(* CODESYS project e!C_Integration_Test_1.ECP

Project tree, tasks and I/O mapping:
  PFC200_CS_2ETH_RS_CAN_DPS : 750-8206 PFC200 2ETH RS CAN DPS, WAGO, order no. 0750-8206, version 5.11.1.16
    application PFC8206
      libraries: Util, * (System); VisuDialogs, * (System)
      task PLC_Task (cyclic, interval t#10ms, priority 14) calls PLC_PRG
      task VISU_TASK (cyclic, interval 100 ms, priority 15) calls VisuElems.Visu_Prg
      task AlarmManagerTask (cyclic, interval 50 ms, priority 15) calls AlarmManager.Alarm_Prg
      program PLC_PRG [ST]: BlinkTest1, Modbus, NetVar
      visualisation Visu1
      Alarm_Configuration
        alarm class Error (priority 10, acknowledge REP_ACK)
        alarm class Warning (priority 30, acknowledge REP)
        alarm class Info (priority 100, acknowledge REP)
        AlarmStorage
        text list AlarmGroup1
        alarm group AlarmGroup1
            0 [Error]: Comparison Equal, ExpressionToCompare TRUE, Expression DO1 - "MinAlarm1"
      Scaling/
        function block fbScale_AI_455 [ST]
        function block fbScale_AI_457 [ST]
        function block fbScale_AI_457_Positiv [ST]
        function block fbScale_AI_460 [ST]
        function block fbScale_AI_461 [ST]
        function block fbScale_AI_466 [ST]
        function block fbScale_AI_473 [ST]
        function block fbScale_AO_552 [ST]
        function block fbScale_AO_555 [ST]
        function block fbScale_AO_556 [ST]
        function block fbScale_AO_559 [ST]
      program ScaleTest [CFC]: AnalogInput, AnalogOutput
      MODBUS/
        data type typFC352_tcp
        data type typPFC200_CS_2ETH_CAN_tcpPFC8203PLC_PRG
        data type typPFC200_CS_2ETH_CAN_tcpPFC8203
        data type typPFC200_CS_2ETH_CAN_tcp
      global variables MODBUS
      global variables NVL1_From_8206
      declarations NVL1_From_8203
    DeviceAdapter
    CANbus
      WAGO_CANopen_Manager : WAGO CANopen Manager, WAGO, version 3.5.4.10
          settings: ConfigVersion = 50659584
        _750_347m_V14 : 750-347m_V14, WAGO, order no. 750-347, version Revision=16#00000001, FileVersion=1.14
            settings: General Options.Reset Node = false; NODEIDSAVED = 5; SDO Timeout = 1000000; SubIndex for reset node = 0; Emergency-General Parameters.Emergency COBID = 16#00000085; Settings.COBID = 16#00000205; Settings.Transmission Type = 16#FF; Settings.available PDO-Parameter.Inhibit Time available = FALSE; Settings.available PDO-Parameter.Event Timer available = FALSE; Settings.Inhibit Time = 0; Settings.Event Timer = 0; Generic COBID = '$NODEID+16#0200'; Process by CANopenManager = TRUE; Settings.COBID = 16#00000185; Settings.Transmission Type = 16#FF; Settings.available PDO-Parameter.Inhibit Time available = TRUE; Settings.available PDO-Parameter.Event Timer available = TRUE; Settings.Inhibit Time = 0; Settings.Event Timer = 0; Generic COBID = '$NODEID+16#0180'; Process by CANopenManager = TRUE; N/A.Index = 16#6200; N/A.Subindex = 16#01; N/A.ObjectLength = 8; N/A.Index = 16#6401; N/A.Subindex = 16#01; N/A.ObjectLength = 16; N/A.Index = 16#6401; N/A.Subindex = 16#02; N/A.ObjectLength = 16; N/A.Index = 16#6401; N/A.Subindex = 16#03; N/A.ObjectLength = 16; N/A.Index = 16#6401; N/A.Subindex = 16#04; N/A.ObjectLength = 16; SDO List.Set Guardtime.Index = 16#100C; SDO List.Set Guardtime.Subindex = 16#00; SDO List.Set Guardtime.Value = 16#00000000; SDO List.Set Guardtime.Size = 16;
              SDO List.Set Guardtime.AbortIfError = FALSE; SDO List.Set Guardtime.JumpToLine = FALSE; SDO List.Set Guardtime.Line = 0; SDO List.Set Lifetime.Index = 16#100D; SDO List.Set Lifetime.Subindex = 16#00; SDO List.Set Lifetime.Value = 16#00000000; SDO List.Set Lifetime.Size = 8; SDO List.Set Lifetime.AbortIfError = FALSE; SDO List.Set Lifetime.JumpToLine = FALSE; SDO List.Set Lifetime.Line = 0; SDO List.Disable Emcy CobID.Index = 16#1014; SDO List.Disable Emcy CobID.Subindex = 16#00; SDO List.Disable Emcy CobID.Value = 16#80000085; SDO List.Disable Emcy CobID.Size = 32; SDO List.Disable Emcy CobID.AbortIfError = FALSE; SDO List.Disable Emcy CobID.JumpToLine = FALSE; SDO List.Disable Emcy CobID.Line = 0; SDO List.Set Emcy CobID.Index = 16#1014; SDO List.Set Emcy CobID.Subindex = 16#00; SDO List.Set Emcy CobID.Value = 16#00000085; SDO List.Set Emcy CobID.Size = 32; SDO List.Set Emcy CobID.AbortIfError = FALSE; SDO List.Set Emcy CobID.JumpToLine = FALSE; SDO List.Set Emcy CobID.Line = 0; SDO List.Set Heartbeat Consumer.Index = 16#1016; SDO List.Set Heartbeat Consumer.Subindex = 16#01; SDO List.Set Heartbeat Consumer.Value = 0; SDO List.Set Heartbeat Consumer.Size = 32; SDO List.Set Heartbeat Consumer.AbortIfError = FALSE; SDO List.Set Heartbeat Consumer.JumpToLine = FALSE; SDO List.Set Heartbeat Consumer.Line = 0; SDO List.Set Heartbeat Consumer.Index = 16#1016; SDO List.Set Heartbeat Consumer.Subindex = 16#02; SDO List.Set Heartbeat Consumer.Value = 0; SDO List.Set Heartbeat Consumer.Size = 32; SDO List.Set Heartbeat Consumer.AbortIfError = FALSE; SDO List.Set Heartbeat Consumer.JumpToLine = FALSE; SDO List.Set Heartbeat Consumer.Line = 0; SDO List.Set Heartbeat Consumer.Index = 16#1016; SDO List.Set Heartbeat Consumer.Subindex = 16#03;
              SDO List.Set Heartbeat Consumer.Value = 0; SDO List.Set Heartbeat Consumer.Size = 32; SDO List.Set Heartbeat Consumer.AbortIfError = FALSE; SDO List.Set Heartbeat Consumer.JumpToLine = FALSE; SDO List.Set Heartbeat Consumer.Line = 0; SDO List.Set Heartbeat Consumer.Index = 16#1016; SDO List.Set Heartbeat Consumer.Subindex = 16#04; SDO List.Set Heartbeat Consumer.Value = 0; SDO List.Set Heartbeat Consumer.Size = 32; SDO List.Set Heartbeat Consumer.AbortIfError = FALSE; SDO List.Set Heartbeat Consumer.JumpToLine = FALSE; SDO List.Set Heartbeat Consumer.Line = 0; SDO List.Set Heartbeat Consumer.Index = 16#1016; SDO List.Set Heartbeat Consumer.Subindex = 16#05; SDO List.Set Heartbeat Consumer.Value = 0; SDO List.Set Heartbeat Consumer.Size = 32; SDO List.Set Heartbeat Consumer.AbortIfError = FALSE; SDO List.Set Heartbeat Consumer.JumpToLine = FALSE; SDO List.Set Heartbeat Consumer.Line = 0; SDO List.Set Heartbeat Producer.Index = 16#1017; SDO List.Set Heartbeat Producer.Subindex = 16#00; SDO List.Set Heartbeat Producer.Value = 16#00000000; SDO List.Set Heartbeat Producer.Size = 16; SDO List.Set Heartbeat Producer.AbortIfError = FALSE; SDO List.Set Heartbeat Producer.JumpToLine = FALSE; SDO List.Set Heartbeat Producer.Line = 0; SDO List.Disable PDO.Index = 16#1400; SDO List.Disable PDO.Subindex = 16#01; SDO List.Disable PDO.Value = 16#80000205; SDO List.Disable PDO.Size = 32; SDO List.Disable PDO.AbortIfError = FALSE; SDO List.Disable PDO.JumpToLine = FALSE; SDO List.Disable PDO.Line = 0; SDO List.Set transmission type.Index = 16#1400; SDO List.Set transmission type.Subindex = 16#02; SDO List.Set transmission type.Value = 16#FF; SDO List.Set transmission type.Size = 8; SDO List.Set transmission type.AbortIfError = FALSE; SDO List.Set transmission type.JumpToLine = FALSE; SDO List.Set transmission type.Line = 0;
              SDO List.Clear pdo mapping.Index = 16#1600; SDO List.Clear pdo mapping.Subindex = 16#00; SDO List.Clear pdo mapping.Value = 16#0; SDO List.Clear pdo mapping.Size = 8; SDO List.Clear pdo mapping.AbortIfError = FALSE; SDO List.Clear pdo mapping.JumpToLine = FALSE; SDO List.Clear pdo mapping.Line = 0; SDO List.Set Mapping.Index = 16#1600; SDO List.Set Mapping.Subindex = 16#01; SDO List.Set Mapping.Value = 16#62000108; SDO List.Set Mapping.Size = 32; SDO List.Set Mapping.AbortIfError = FALSE; SDO List.Set Mapping.JumpToLine = FALSE; SDO List.Set Mapping.Line = 0; SDO List.Set number of mappings.Index = 16#1600; SDO List.Set number of mappings.Subindex = 16#00; SDO List.Set number of mappings.Value = 16#01; SDO List.Set number of mappings.Size = 8; SDO List.Set number of mappings.AbortIfError = FALSE; SDO List.Set number of mappings.JumpToLine = FALSE; SDO List.Set number of mappings.Line = 0; SDO List.Set and enable COB-ID.Index = 16#1400; SDO List.Set and enable COB-ID.Subindex = 16#01; SDO List.Set and enable COB-ID.Value = 16#00000205; SDO List.Set and enable COB-ID.Size = 32; SDO List.Set and enable COB-ID.AbortIfError = FALSE; SDO List.Set and enable COB-ID.JumpToLine = FALSE; SDO List.Set and enable COB-ID.Line = 0; SDO List.Disable PDO.Index = 16#1800; SDO List.Disable PDO.Subindex = 16#01; SDO List.Disable PDO.Value = 16#80000185; SDO List.Disable PDO.Size = 32; SDO List.Disable PDO.AbortIfError = FALSE; SDO List.Disable PDO.JumpToLine = FALSE; SDO List.Disable PDO.Line = 0; SDO List.Set transmission type.Index = 16#1800; SDO List.Set transmission type.Subindex = 16#02; SDO List.Set transmission type.Value = 16#FF; SDO List.Set transmission type.Size = 8; SDO List.Set transmission type.AbortIfError = FALSE;
              SDO List.Set transmission type.JumpToLine = FALSE; SDO List.Set transmission type.Line = 0; SDO List.Set inhibit time.Index = 16#1800; SDO List.Set inhibit time.Subindex = 16#03; SDO List.Set inhibit time.Value = 16#0000; SDO List.Set inhibit time.Size = 16; SDO List.Set inhibit time.AbortIfError = FALSE; SDO List.Set inhibit time.JumpToLine = FALSE; SDO List.Set inhibit time.Line = 0; SDO List.Set event time.Index = 16#1800; SDO List.Set event time.Subindex = 16#05; SDO List.Set event time.Value = 16#0000; SDO List.Set event time.Size = 16; SDO List.Set event time.AbortIfError = FALSE; SDO List.Set event time.JumpToLine = FALSE; SDO List.Set event time.Line = 0; SDO List.Clear pdo mapping.Index = 16#1A00; SDO List.Clear pdo mapping.Subindex = 16#00; SDO List.Clear pdo mapping.Value = 16#0; SDO List.Clear pdo mapping.Size = 8; SDO List.Clear pdo mapping.AbortIfError = FALSE; SDO List.Clear pdo mapping.JumpToLine = FALSE; SDO List.Clear pdo mapping.Line = 0; SDO List.Set Mapping.Index = 16#1A00; SDO List.Set Mapping.Subindex = 16#01; SDO List.Set Mapping.Value = 16#64010110; SDO List.Set Mapping.Size = 32; SDO List.Set Mapping.AbortIfError = FALSE; SDO List.Set Mapping.JumpToLine = FALSE; SDO List.Set Mapping.Line = 0; SDO List.Set Mapping.Index = 16#1A00; SDO List.Set Mapping.Subindex = 16#02; SDO List.Set Mapping.Value = 16#64010210; SDO List.Set Mapping.Size = 32; SDO List.Set Mapping.AbortIfError = FALSE; SDO List.Set Mapping.JumpToLine = FALSE; SDO List.Set Mapping.Line = 0; SDO List.Set Mapping.Index = 16#1A00; SDO List.Set Mapping.Subindex = 16#03; SDO List.Set Mapping.Value = 16#64010310;
              SDO List.Set Mapping.Size = 32; SDO List.Set Mapping.AbortIfError = FALSE; SDO List.Set Mapping.JumpToLine = FALSE; SDO List.Set Mapping.Line = 0; SDO List.Set Mapping.Index = 16#1A00; SDO List.Set Mapping.Subindex = 16#04; SDO List.Set Mapping.Value = 16#64010410; SDO List.Set Mapping.Size = 32; SDO List.Set Mapping.AbortIfError = FALSE; SDO List.Set Mapping.JumpToLine = FALSE; SDO List.Set Mapping.Line = 0; SDO List.Set number of mappings.Index = 16#1A00; SDO List.Set number of mappings.Subindex = 16#00; SDO List.Set number of mappings.Value = 16#04; SDO List.Set number of mappings.Size = 8; SDO List.Set number of mappings.AbortIfError = FALSE; SDO List.Set number of mappings.JumpToLine = FALSE; SDO List.Set number of mappings.Line = 0; SDO List.Set and enable COB-ID.Index = 16#1800; SDO List.Set and enable COB-ID.Subindex = 16#01; SDO List.Set and enable COB-ID.Value = 16#00000185; SDO List.Set and enable COB-ID.Size = 32; SDO List.Set and enable COB-ID.AbortIfError = FALSE; SDO List.Set and enable COB-ID.JumpToLine = FALSE; SDO List.Set and enable COB-ID.Line = 0; ConfigVersion = 50659584
          DeviceAdapter
          _75x_504_1 : 75x-504, WAGO, order no. 75x-504, version Revision=16#00000001, FileVersion=1.14
              settings: Number of Params = 1; WriteOutput8Bit : _75x_504_1.Index = 16#6200; WriteOutput8Bit : _75x_504_1.Subindex = 16#01; WriteOutput8Bit : _75x_504_1.Startbit = 0; WriteOutput8Bit : _75x_504_1.Endbit = 3
              output PFC8206.PLC_PRG.BLINK_1.OUT : BOOL  // WriteOutput8Bit : _75x_504.WriteOutput8Bit : _75x_504
              unmapped channels: WriteOutput8Bit : _75x_504
          _75x_455_1 : 75x-455, WAGO, order no. 75x-455, version Revision=16#00000001, FileVersion=1.14
              settings: Number of Params = 4; ReadAnalogueInput16Bit : _75x_455_1.Index = 16#6401; ReadAnalogueInput16Bit : _75x_455_1.Subindex = 16#01; ReadAnalogueInput16Bit : _75x_455_1.Startbit = 0; ReadAnalogueInput16Bit : _75x_455_1.Endbit = 15; ReadAnalogueInput16Bit : _75x_455_1.Index = 16#6401; ReadAnalogueInput16Bit : _75x_455_1.Subindex = 16#02; ReadAnalogueInput16Bit : _75x_455_1.Startbit = 0; ReadAnalogueInput16Bit : _75x_455_1.Endbit = 15; ReadAnalogueInput16Bit : _75x_455_1.Index = 16#6401; ReadAnalogueInput16Bit : _75x_455_1.Subindex = 16#03; ReadAnalogueInput16Bit : _75x_455_1.Startbit = 0; ReadAnalogueInput16Bit : _75x_455_1.Endbit = 15; ReadAnalogueInput16Bit : _75x_455_1.Index = 16#6401; ReadAnalogueInput16Bit : _75x_455_1.Subindex = 16#04; ReadAnalogueInput16Bit : _75x_455_1.Startbit = 0; ReadAnalogueInput16Bit : _75x_455_1.Endbit = 15
              unmapped channels: ReadAnalogueInput16Bit : _75x_455_1, ReadAnalogueInput16Bit : _75x_455_1, ReadAnalogueInput16Bit : _75x_455_1, ReadAnalogueInput16Bit : _75x_455_1
    Serial
      COM1 : COM1, WAGO, version 0.0.0.19
    PROFIBUS
      PROFIBUS : PROFIBUS, WAGO, version 1.0.0.0 (disabled)
    Kbus : Kbus, WAGO, version 1.4.0.2
        unmapped channels: K-BUS diagnostics
      _8_DO_DI_Generic : 075x-8DO8DI, WAGO, order no. 075x-8DO8DI, version 0.0.0.13
          settings: K-BUS Module slot index = 1
          output DO1 : BOOL  // _OUT._OUT
          unmapped channels: _IN, _OUT
        DeviceAdapter
      _4_AI_10V_DC_s_e : 0750-0457, WAGO, order no. 0750-0457, version 0.0.0.9
          settings: K-BUS Module slot index = 3
          input  AI_457_1_1 : WORD  // _IW 1
          unmapped channels: _IW 2, _IW 3, _IW 4
        DeviceAdapter
      _4_AO_0_10V_DC : 0750-0559, WAGO, order no. 0750-0559, version 0.0.0.13
          settings: K-BUS Module slot index = 2
          output AO_559_1_1 : WORD  // _QW 1
          unmapped channels: _QW 2, _QW 3, _QW 4
        DeviceAdapter
    MODBUS
      MODBUS : MODBUS, WAGO, order no. n/a, version 1.1.1.15
        _internal_1006_0001_Master : MODBUS Master, WAGO, order no. n/a, version 1.1.1.15
          _internal_1006_0001_IP : MODBUS IP Interface, WAGO, order no. n/a, version 1.1.1.15
              settings: IP settings.Address = '192.168.1.8'; Minimum Request Interval = 0 ms
            _internal_1006_0001_Remote_Slave : MODBUS Remote Slave, WAGO, order no. n/a, version 1.1.1.15
                settings: GeneratedChannel 100005.Cycle Time = 200 ms; GeneratedChannel 100005.Write Address = 512 Registers or Coils; GeneratedChannel 100005.Write Length = 2 Registers or Coils; Offset 100010 = 0; Offset 100030 = 1; Slave address / Unit identifier = 1
                output PFC8206.MODBUS.FC352_tcp.dOut_1 : BOOL  // Mapping100020
                output PFC8206.MODBUS.FC352_tcp.dOut_2 : BOOL  // Mapping100040
          _internal_1006_0001_IP_1 : MODBUS IP Interface, WAGO, order no. n/a, version 1.1.1.15
              settings: IP settings.Address = '192.168.1.118'; Minimum Request Interval = 0 ms
            _internal_1006_0001_Remote_Slave_1 : MODBUS Remote Slave, WAGO, order no. n/a, version 1.1.1.15
                settings: GeneratedChannel 100005.Cycle Time = 200 ms; GeneratedChannel 100005.Read Length = 1 Registers or Coils; GeneratedChannel 100005.Write Address = 32000 Registers or Coils; GeneratedChannel 100005.Write Length = 1 Registers or Coils; Offset 100010 = 0; Offset 100030 = 0; Slave address / Unit identifier = 1
                input  PFC8206.MODBUS.PFC200_CS_2ETH_CAN_tcp.PFC8203.PLC_PRG.wMbVar1_From_8203 : WORD  // Mapping100020
                output PFC8206.MODBUS.PFC200_CS_2ETH_CAN_tcp.PFC8203.PLC_PRG.wMbVar1_To_8203 : WORD  // Mapping100040
  FC352 : 750-352, WAGO, order no. 0750-0352, version 0.0.0.9
    DeviceAdapter
    Kbus : Kbus, WAGO, version 0.0.0.101
      _2_DO_Generic : 075x-2DO, WAGO, order no. 075x-2DO, version 0.0.0.13
          settings: K-BUS Module slot index = 1
          unmapped channels: _OUT
        DeviceAdapter
  PFC200_CS_2ETH_CAN : 750-8203 PFC200 2ETH CAN, WAGO, order no. 0750-8203, version 5.11.1.16
    application PFC8203
      libraries: 
      task PLC_Task (cyclic, interval t#10ms, priority 14) calls PLC_PRG
      program PLC_PRG [ST]: NetVar, Modbus
      declarations NVL1_From_8206
      global variables NVL1_From_8203
      Symbols
    DeviceAdapter
    CANbus
    MODBUS
      MODBUS : MODBUS, WAGO, order no. n/a, version 1.1.1.15
        LocalDeviceModbus : MODBUS Slave, WAGO, order no. n/a, version 1.1.1.15
            settings: OffsetMap = 0; OffsetMap = 0
            output PFC8203.PLC_PRG.wMbVar1_From_8203 : WORD  // 
            input  PFC8203.PLC_PRG.wMbVar1_To_8203 : WORD  // 
          TcpSettings : Modbus TCP Slave, WAGO, order no. n/a, version 1.1.1.15
    Kbus : Kbus, WAGO, version 1.4.0.2
        unmapped channels: K-BUS diagnostics
      _8_DO_DI_Generic : 075x-8DO8DI, WAGO, order no. 075x-8DO8DI, version 0.0.0.13
          settings: K-BUS Module slot index = 1
          unmapped channels: _IN, _OUT
        DeviceAdapter
  libraries: VisuSymbols, 3.5.10.0 (System); WagoVisuIcons, 1.0.0.8 (WAGO)
  text list GlobalTextList
*)

// PFC200_CS_2ETH_RS_CAN_DPS/PFC8206/MODBUS/typFC352_tcp
TYPE typFC352_tcp:
STRUCT
	dOut_1: BOOL;
	dOut_2: BOOL;
END_STRUCT
END_TYPE

// PFC200_CS_2ETH_RS_CAN_DPS/PFC8206/MODBUS/typPFC200_CS_2ETH_CAN_tcpPFC8203PLC_PRG
TYPE typPFC200_CS_2ETH_CAN_tcpPFC8203PLC_PRG:
STRUCT
	wMbVar1_From_8203: WORD;
	wMbVar1_To_8203: WORD;
END_STRUCT
END_TYPE

// PFC200_CS_2ETH_RS_CAN_DPS/PFC8206/MODBUS/typPFC200_CS_2ETH_CAN_tcpPFC8203
TYPE typPFC200_CS_2ETH_CAN_tcpPFC8203:
STRUCT
	PLC_PRG: typPFC200_CS_2ETH_CAN_tcpPFC8203PLC_PRG;
END_STRUCT
END_TYPE

// PFC200_CS_2ETH_RS_CAN_DPS/PFC8206/MODBUS/typPFC200_CS_2ETH_CAN_tcp
TYPE typPFC200_CS_2ETH_CAN_tcp:
STRUCT
	PFC8203: typPFC200_CS_2ETH_CAN_tcpPFC8203;
END_STRUCT
END_TYPE

// PFC200_CS_2ETH_RS_CAN_DPS/PFC8206/MODBUS
VAR_GLOBAL
	FC352_tcp: typFC352_tcp;
	PFC200_CS_2ETH_CAN_tcp: typPFC200_CS_2ETH_CAN_tcp;
END_VAR

// PFC200_CS_2ETH_RS_CAN_DPS/PFC8206/NVL1_From_8206
VAR_GLOBAL
	wNetVar1From8206 : WORD;
END_VAR

// PFC200_CS_2ETH_CAN/PFC8203/NVL1_From_8206
//This gobal variable list is received via the network.
//Sender: NVL1_From_8206 [PFC200_CS_2ETH_RS_CAN_DPS: PLC Logic: PFC8206]
//Protocol: UDP

VAR_GLOBAL
	wNetVar1From8206 : WORD;
END_VAR

// PFC200_CS_2ETH_CAN/PFC8203/NVL1_From_8203
VAR_GLOBAL
	wNetVar1From8203 : WORD;
END_VAR

// PFC200_CS_2ETH_RS_CAN_DPS/PFC8206/NVL1_From_8203
//This gobal variable list is received via the network.
//Sender: NVL1_From_8203 [PFC200_CS_2ETH_CAN: PLC Logic: PFC8203]
//Protocol: UDP

VAR_GLOBAL
	wNetVar1From8203 : WORD;
END_VAR

// PFC200_CS_2ETH_CAN/PFC8203/PLC_PRG
PROGRAM PLC_PRG
VAR
	
	wMbVar1_To_8203: WORD;	
	wMbVar1_From_8203: WORD;
END_VAR



NetVar();
Modbus();

ACTION NetVar:

wNetVar1From8203 := wNetVar1From8203 + 1;
wNetVar1From8206;
END_ACTION

ACTION Modbus:


wMbVar1_From_8203 := wMbVar1_From_8203 + 1;
wMbVar1_To_8203;
END_ACTION

END_PROGRAM

// PFC200_CS_2ETH_RS_CAN_DPS/PFC8206/PLC_PRG
PROGRAM PLC_PRG
VAR
	BLINK_1: BLINK;
	tTimeLow: TIME := T#5S;
	tTimeHigh: TIME := T#1S;
END_VAR



BlinkTest1();
ScaleTest();
Modbus();
NetVar();

ACTION BlinkTest1:
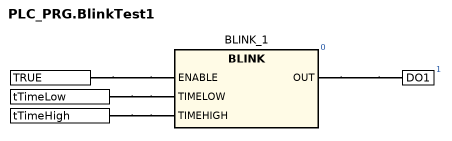
BLINK_1(ENABLE := TRUE, TIMELOW := tTimeLow, TIMEHIGH := tTimeHigh); // BLINK
DO1 := BLINK_1.OUT;
END_ACTION

ACTION Modbus:



FC352_tcp.dOut_1 := BLINK_1.OUT;

PFC200_CS_2ETH_CAN_tcp.PFC8203.PLC_PRG.wMbVar1_From_8203;
PFC200_CS_2ETH_CAN_tcp.PFC8203.PLC_PRG.wMbVar1_To_8203 := PFC200_CS_2ETH_CAN_tcp.PFC8203.PLC_PRG.wMbVar1_To_8203 + 1;
END_ACTION

ACTION NetVar:


wNetVar1From8206 := wNetVar1From8206 + 1;
wNetVar1From8203;
END_ACTION

END_PROGRAM

// PFC200_CS_2ETH_RS_CAN_DPS/PFC8206/ScaleTest
PROGRAM ScaleTest
VAR

	Scale_AI_Pressure_1: fbScale_AI_455;
	Scale_AI_Distance_1: fbScale_AI_473;
	Scale_AI_Level_1: fbScale_AI_466;
	Scale_AI_Temp_1: fbScale_AI_460;
	Scale_AI_EngineTemp_1: fbScale_AI_461;
	Scale_AI_SpeedActual_1: fbScale_AI_457_Positiv;
	Scale_AO_SpeedSet_1: fbScale_AO_559;
	Scale_AO_PressureSet_1: fbScale_AO_555;
	Scale_AO_LevelSet_1: fbScale_AO_556;
	Scale_AO_DistanceSet_1: fbScale_AO_552;

	AI_Pressure_1_Signal: REAL;
	AI_Pressure_1_SignalStatus : BYTE;
	AI_Distance_1_Signal: REAL;
	AI_Distance_1_SignalStatus : BYTE;
	AI_Level_1_Signal: REAL;
	AI_Level_1_SignalStatus : BYTE;
	AI_Temp_1_Signal: REAL;
	AI_Temp_1_SignalStatus : BYTE;
	AI_EngineTemp_1_Signal: REAL;
	AI_EngineTemp_1_SignalStatus : BYTE;
	AI_SpeedActual_1_Signal: REAL;
	AI_SpeedActual_1_SignalStatus: BYTE;
	AO_SpeedSet_1_Signal: REAL;
	AO_SpeedSet_1_SignalStatus: BYTE;
	AO_PressureSet_1_Signal: REAL;
	AO_PressureSet_1_SignalStatus: BYTE;
	AO_LevelSet_1_Signal: REAL;
	AO_LevelSet_1_SignalStatus: BYTE;
	AO_DistanceSet_1_Signal: REAL;
	AO_DistanceSet_1_SignalStatus: BYTE;

	AO_552_1_1_sim: WORD;
	AO_555_1_1_sim: WORD;
	AO_556_1_1_sim: WORD;
	AI_455_1_1_sim: WORD;
	AI_473_1_1_sim: WORD;
	AI_466_1_1_sim: WORD;
	AI_460_1_1_sim: WORD;
	AI_461_1_1_sim: WORD;

END_VAR

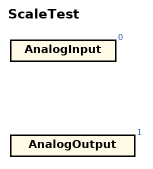
AnalogInput();
AnalogOutput();

ACTION AnalogInput:
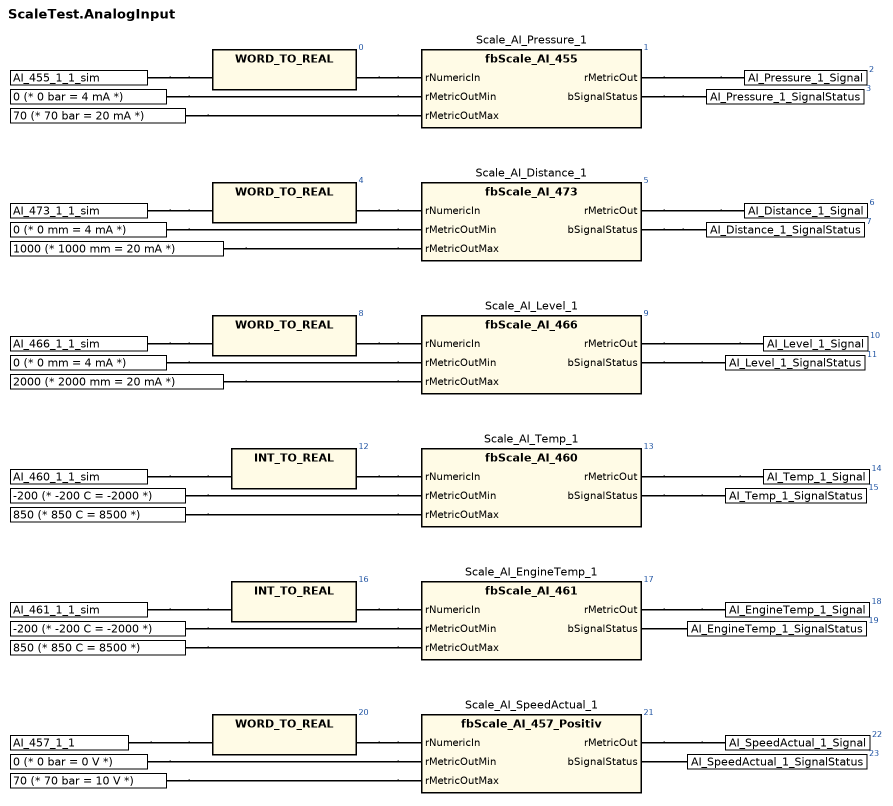
Scale_AI_Pressure_1(
    rNumericIn := WORD_TO_REAL(AI_455_1_1_sim),
    rMetricOutMin := 0 (* 0 bar = 4 mA *),
    rMetricOutMax := 70 (* 70 bar = 20 mA *)); // fbScale_AI_455
AI_Pressure_1_Signal := Scale_AI_Pressure_1.rMetricOut;
AI_Pressure_1_SignalStatus := Scale_AI_Pressure_1.bSignalStatus;
Scale_AI_Distance_1(
    rNumericIn := WORD_TO_REAL(AI_473_1_1_sim),
    rMetricOutMin := 0 (* 0 mm = 4 mA *),
    rMetricOutMax := 1000 (* 1000 mm = 20 mA *)); // fbScale_AI_473
AI_Distance_1_Signal := Scale_AI_Distance_1.rMetricOut;
AI_Distance_1_SignalStatus := Scale_AI_Distance_1.bSignalStatus;
Scale_AI_Level_1(
    rNumericIn := WORD_TO_REAL(AI_466_1_1_sim),
    rMetricOutMin := 0 (* 0 mm = 4 mA *),
    rMetricOutMax := 2000 (* 2000 mm = 20 mA *)); // fbScale_AI_466
AI_Level_1_Signal := Scale_AI_Level_1.rMetricOut;
AI_Level_1_SignalStatus := Scale_AI_Level_1.bSignalStatus;
Scale_AI_Temp_1(
    rNumericIn := INT_TO_REAL(AI_460_1_1_sim),
    rMetricOutMin := -200 (* -200 C = -2000 *),
    rMetricOutMax := 850 (* 850 C = 8500 *)); // fbScale_AI_460
AI_Temp_1_Signal := Scale_AI_Temp_1.rMetricOut;
AI_Temp_1_SignalStatus := Scale_AI_Temp_1.bSignalStatus;
Scale_AI_EngineTemp_1(
    rNumericIn := INT_TO_REAL(AI_461_1_1_sim),
    rMetricOutMin := -200 (* -200 C = -2000 *),
    rMetricOutMax := 850 (* 850 C = 8500 *)); // fbScale_AI_461
AI_EngineTemp_1_Signal := Scale_AI_EngineTemp_1.rMetricOut;
AI_EngineTemp_1_SignalStatus := Scale_AI_EngineTemp_1.bSignalStatus;
Scale_AI_SpeedActual_1(
    rNumericIn := WORD_TO_REAL(AI_457_1_1),
    rMetricOutMin := 0 (* 0 bar = 0 V *),
    rMetricOutMax := 70 (* 70 bar = 10 V *)); // fbScale_AI_457_Positiv
AI_SpeedActual_1_Signal := Scale_AI_SpeedActual_1.rMetricOut;
AI_SpeedActual_1_SignalStatus := Scale_AI_SpeedActual_1.bSignalStatus;
END_ACTION

ACTION AnalogOutput:
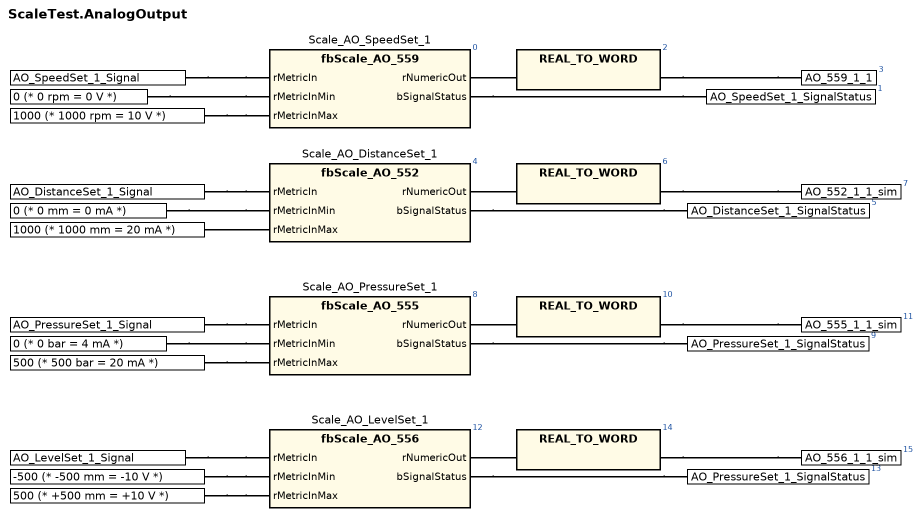
Scale_AO_SpeedSet_1(
    rMetricIn := AO_SpeedSet_1_Signal,
    rMetricInMin := 0 (* 0 rpm = 0 V *),
    rMetricInMax := 1000 (* 1000 rpm = 10 V *)); // fbScale_AO_559
AO_SpeedSet_1_SignalStatus := Scale_AO_SpeedSet_1.bSignalStatus;
AO_559_1_1 := REAL_TO_WORD(Scale_AO_SpeedSet_1.rNumericOut);
Scale_AO_DistanceSet_1(
    rMetricIn := AO_DistanceSet_1_Signal,
    rMetricInMin := 0 (* 0 mm = 0 mA *),
    rMetricInMax := 1000 (* 1000 mm = 20 mA *)); // fbScale_AO_552
AO_DistanceSet_1_SignalStatus := Scale_AO_DistanceSet_1.bSignalStatus;
AO_552_1_1_sim := REAL_TO_WORD(Scale_AO_DistanceSet_1.rNumericOut);
Scale_AO_PressureSet_1(
    rMetricIn := AO_PressureSet_1_Signal,
    rMetricInMin := 0 (* 0 bar = 4 mA *),
    rMetricInMax := 500 (* 500 bar = 20 mA *)); // fbScale_AO_555
AO_PressureSet_1_SignalStatus := Scale_AO_PressureSet_1.bSignalStatus;
AO_555_1_1_sim := REAL_TO_WORD(Scale_AO_PressureSet_1.rNumericOut);
Scale_AO_LevelSet_1(
    rMetricIn := AO_LevelSet_1_Signal,
    rMetricInMin := -500 (* -500 mm = -10 V *),
    rMetricInMax := 500 (* +500 mm = +10 V *)); // fbScale_AO_556
AO_PressureSet_1_SignalStatus := Scale_AO_LevelSet_1.bSignalStatus;
AO_556_1_1_sim := REAL_TO_WORD(Scale_AO_LevelSet_1.rNumericOut);
END_ACTION

END_PROGRAM

// PFC200_CS_2ETH_RS_CAN_DPS/PFC8206/Scaling/fbScale_AI_455
FUNCTION_BLOCK fbScale_AI_455

VAR_INPUT

	rNumericIn: REAL;
	rMetricOutMin: REAL := 4;
	rMetricOutMax: REAL := 20;

END_VAR


VAR_OUTPUT

	rMetricOut: REAL;
	bSignalStatus : BYTE;

END_VAR


VAR

	LIN_TRAFO_ScaleAnalog: LIN_TRAFO;
	rNumericInMin: REAL := 0;
	rNumericInMax: REAL := 32760;

END_VAR



LIN_TRAFO_ScaleAnalog(
	IN			:= rNumericIn,
	IN_MIN		:= rNumericInMin,
	IN_MAX		:= rNumericInMax,
	OUT_MIN		:= rMetricOutMin,
	OUT_MAX		:= rMetricOutMax,
	OUT			=> rMetricOut );


IF ( (REAL_TO_WORD(rNumericIn) AND 16#0003) > 0 ) THEN
	IF (REAL_TO_WORD(rNumericIn) > rNumericInMax) THEN
		rMetricOut := rMetricOutMax;
		bSignalStatus := 2;
	ELSE
		rMetricOut := rMetricOutMin;
		bSignalStatus := 1;
	END_IF
ELSE
	bSignalStatus := 0;
END_IF

END_FUNCTION_BLOCK

// PFC200_CS_2ETH_RS_CAN_DPS/PFC8206/Scaling/fbScale_AI_473
FUNCTION_BLOCK fbScale_AI_473

VAR_INPUT

	rNumericIn: REAL;
	rMetricOutMin: REAL := 4;
	rMetricOutMax: REAL := 20;

END_VAR


VAR_OUTPUT

	rMetricOut: REAL;
	bSignalStatus : BYTE;

END_VAR


VAR

	LIN_TRAFO_ScaleAnalog: LIN_TRAFO;
	rNumericInMin: REAL := 4096;
	rNumericInMax: REAL := 20480;

END_VAR



LIN_TRAFO_ScaleAnalog(
	IN			:= rNumericIn,
	IN_MIN		:= rNumericInMin,
	IN_MAX		:= rNumericInMax,
	OUT_MIN		:= rMetricOutMin,
	OUT_MAX		:= rMetricOutMax,
	OUT			=> rMetricOut );


IF ( (REAL_TO_WORD(rNumericIn) AND 16#0003) > 0 ) THEN
	IF (REAL_TO_WORD(rNumericIn) > rNumericInMax) THEN
		rMetricOut := rMetricOutMax;
		bSignalStatus := 2;
	ELSE
		rMetricOut := rMetricOutMin;
		bSignalStatus := 1;
	END_IF
ELSE
	bSignalStatus := 0;
END_IF

END_FUNCTION_BLOCK

// PFC200_CS_2ETH_RS_CAN_DPS/PFC8206/Scaling/fbScale_AI_466
FUNCTION_BLOCK fbScale_AI_466

VAR_INPUT

	rNumericIn: REAL;
	rMetricOutMin: REAL := 4;
	rMetricOutMax: REAL := 20;

END_VAR


VAR_OUTPUT

	rMetricOut: REAL;
	bSignalStatus : BYTE;

END_VAR


VAR

	LIN_TRAFO_ScaleAnalog: LIN_TRAFO;
	rNumericInMin: REAL := 0;
	rNumericInMax: REAL := 32760;

END_VAR



LIN_TRAFO_ScaleAnalog(
	IN			:= rNumericIn,
	IN_MIN		:= rNumericInMin,
	IN_MAX		:= rNumericInMax,
	OUT_MIN		:= rMetricOutMin,
	OUT_MAX		:= rMetricOutMax,
	OUT			=> rMetricOut );


IF ( (REAL_TO_WORD(rNumericIn) AND 16#0003) > 0 ) THEN
	IF (REAL_TO_WORD(rNumericIn) > rNumericInMax) THEN
		rMetricOut := rMetricOutMax;
		bSignalStatus := 2;
	ELSE
		rMetricOut := rMetricOutMin;
		bSignalStatus := 1;
	END_IF
ELSE
	bSignalStatus := 0;
END_IF

END_FUNCTION_BLOCK

// PFC200_CS_2ETH_RS_CAN_DPS/PFC8206/Scaling/fbScale_AI_460
FUNCTION_BLOCK fbScale_AI_460

VAR_INPUT

	rNumericIn: REAL;
	rMetricOutMin: REAL := -200;
	rMetricOutMax: REAL := 850;

END_VAR


VAR_OUTPUT

	rMetricOut: REAL;
	bSignalStatus : BYTE;

END_VAR


VAR

	LIN_TRAFO_ScaleAnalog: LIN_TRAFO;
	rNumericInMin: REAL := -2000;
	rNumericInMax: REAL := 8500;

END_VAR



LIN_TRAFO_ScaleAnalog(
	IN			:= rNumericIn,
	IN_MIN		:= rNumericInMin,
	IN_MAX		:= rNumericInMax,
	OUT_MIN		:= rMetricOutMin,
	OUT_MAX		:= rMetricOutMax,
	OUT			=> rMetricOut );


IF (rNumericIn >= rNumericInMax) THEN
	rMetricOut := rMetricOutMax;
	bSignalStatus := 1;
ELSIF (rNumericIn < rNumericInMin) THEN
	rMetricOut := rMetricOutMin;
	bSignalStatus := 2;
ELSE
	bSignalStatus := 0;
END_IF

END_FUNCTION_BLOCK

// PFC200_CS_2ETH_RS_CAN_DPS/PFC8206/Scaling/fbScale_AI_461
FUNCTION_BLOCK fbScale_AI_461

VAR_INPUT

	rNumericIn: REAL;
	rMetricOutMin: REAL := -200;
	rMetricOutMax: REAL := 850;

END_VAR


VAR_OUTPUT

	rMetricOut: REAL;
	bSignalStatus : BYTE;

END_VAR


VAR

	LIN_TRAFO_ScaleAnalog: LIN_TRAFO;
	rNumericInMin: REAL := -2000;
	rNumericInMax: REAL := 8500;

END_VAR



LIN_TRAFO_ScaleAnalog(
	IN			:= rNumericIn,
	IN_MIN		:= rNumericInMin,
	IN_MAX		:= rNumericInMax,
	OUT_MIN		:= rMetricOutMin,
	OUT_MAX		:= rMetricOutMax,
	OUT			=> rMetricOut );


IF (rNumericIn >= rNumericInMax) THEN
	rMetricOut := rMetricOutMax;
	bSignalStatus := 1;
ELSIF (rNumericIn < rNumericInMin) THEN
	rMetricOut := rMetricOutMin;
	bSignalStatus := 2;
ELSE
	bSignalStatus := 0;
END_IF

END_FUNCTION_BLOCK

// PFC200_CS_2ETH_RS_CAN_DPS/PFC8206/Scaling/fbScale_AI_457_Positiv
FUNCTION_BLOCK fbScale_AI_457_Positiv

VAR_INPUT

	rNumericIn: REAL;
	rMetricOutMin: REAL := -10;
	rMetricOutMax: REAL := 10;

END_VAR


VAR_OUTPUT

	rMetricOut: REAL;
	bSignalStatus : BYTE;

END_VAR


VAR

	LIN_TRAFO_ScaleAnalog: LIN_TRAFO;
	rNumericInMin: REAL := 0;
	rNumericInMax: REAL := 32760;

END_VAR

LIN_TRAFO_ScaleAnalog(
	IN			:= rNumericIn,
	IN_MIN		:= rNumericInMin,
	IN_MAX		:= rNumericInMax,
	OUT_MIN		:= rMetricOutMin,
	OUT_MAX		:= rMetricOutMax,
	OUT			=> rMetricOut );


IF ( (REAL_TO_WORD(rNumericIn) AND 16#0003) > 0 ) THEN
	IF (REAL_TO_WORD(rNumericIn) > rNumericInMax) THEN
		rMetricOut := rMetricOutMax;
		bSignalStatus := 2;
	ELSE
		rMetricOut := rMetricOutMin;
		bSignalStatus := 1;
	END_IF
ELSE
	bSignalStatus := 0;
END_IF

END_FUNCTION_BLOCK

// PFC200_CS_2ETH_RS_CAN_DPS/PFC8206/Scaling/fbScale_AO_559
FUNCTION_BLOCK fbScale_AO_559

VAR_INPUT

	rMetricIn: REAL;
	rMetricInMin: REAL := 0;
	rMetricInMax: REAL := 10;

END_VAR


VAR_OUTPUT

	rNumericOut: REAL;
	bSignalStatus : BYTE;

END_VAR


VAR

	LIN_TRAFO_ScaleAnalog: LIN_TRAFO;
	rNumericOutMin: REAL := 0;
	rNumericOutMax: REAL := 32767;

END_VAR

LIN_TRAFO_ScaleAnalog(
	IN			:= rMetricIn,
	IN_MIN		:= rMetricInMin,
	IN_MAX		:= rMetricInMax,
	OUT_MIN		:= rNumericOutMin,
	OUT_MAX		:= rNumericOutMax,
	OUT			=> rNumericOut );


IF (rMetricIn > rMetricInMax) THEN
	rNumericOut := rNumericOutMax;
	bSignalStatus := 2;
ELSIF (rMetricIn < rMetricInMin) THEN
	rNumericOut := rNumericOutMin;
	bSignalStatus := 1;
ELSE
	bSignalStatus := 0;
END_IF

END_FUNCTION_BLOCK

// PFC200_CS_2ETH_RS_CAN_DPS/PFC8206/Scaling/fbScale_AO_555
FUNCTION_BLOCK fbScale_AO_555

VAR_INPUT

	rMetricIn: REAL;
	rMetricInMin: REAL := 4;
	rMetricInMax: REAL := 20;

END_VAR


VAR_OUTPUT

	rNumericOut: REAL;
	bSignalStatus : BYTE;

END_VAR


VAR

	LIN_TRAFO_ScaleAnalog: LIN_TRAFO;
	rNumericOutMin: REAL := 0;
	rNumericOutMax: REAL := 32767;

END_VAR

LIN_TRAFO_ScaleAnalog(
	IN			:= rMetricIn,
	IN_MIN		:= rMetricInMin,
	IN_MAX		:= rMetricInMax,
	OUT_MIN		:= rNumericOutMin,
	OUT_MAX		:= rNumericOutMax,
	OUT			=> rNumericOut );


IF (rMetricIn > rMetricInMax) THEN
	rNumericOut := rNumericOutMax;
	bSignalStatus := 2;
ELSIF (rMetricIn < rMetricInMin) THEN
	rNumericOut := rNumericOutMin;
	bSignalStatus := 1;
ELSE
	bSignalStatus := 0;
END_IF

END_FUNCTION_BLOCK

// PFC200_CS_2ETH_RS_CAN_DPS/PFC8206/Scaling/fbScale_AO_556
FUNCTION_BLOCK fbScale_AO_556

VAR_INPUT

	rMetricIn: REAL;
	rMetricInMin: REAL := -10;
	rMetricInMax: REAL := 10;

END_VAR


VAR_OUTPUT

	rNumericOut: REAL;
	bSignalStatus : BYTE;

END_VAR


VAR

	LIN_TRAFO_ScaleAnalog: LIN_TRAFO;
	rNumericOutMin: REAL := -32767;
	rNumericOutMax: REAL := 32767;

END_VAR

LIN_TRAFO_ScaleAnalog(
	IN			:= rMetricIn,
	IN_MIN		:= rMetricInMin,
	IN_MAX		:= rMetricInMax,
	OUT_MIN		:= rNumericOutMin,
	OUT_MAX		:= rNumericOutMax,
	OUT			=> rNumericOut );


IF (rMetricIn > rMetricInMax) THEN
	rNumericOut := rNumericOutMax;
	bSignalStatus := 2;
ELSIF (rMetricIn < rMetricInMin) THEN
	rNumericOut := rNumericOutMin;
	bSignalStatus := 1;
ELSE
	bSignalStatus := 0;
END_IF

END_FUNCTION_BLOCK

// PFC200_CS_2ETH_RS_CAN_DPS/PFC8206/Scaling/fbScale_AO_552
FUNCTION_BLOCK fbScale_AO_552

VAR_INPUT

	rMetricIn: REAL;
	rMetricInMin: REAL := 0;
	rMetricInMax: REAL := 20;

END_VAR


VAR_OUTPUT

	rNumericOut: REAL;
	bSignalStatus : BYTE;

END_VAR


VAR

	LIN_TRAFO_ScaleAnalog: LIN_TRAFO;
	rNumericOutMin: REAL := 0;
	rNumericOutMax: REAL := 32767;

END_VAR

LIN_TRAFO_ScaleAnalog(
	IN			:= rMetricIn,
	IN_MIN		:= rMetricInMin,
	IN_MAX		:= rMetricInMax,
	OUT_MIN		:= rNumericOutMin,
	OUT_MAX		:= rNumericOutMax,
	OUT			=> rNumericOut );


IF (rMetricIn > rMetricInMax) THEN
	rNumericOut := rNumericOutMax;
	bSignalStatus := 2;
ELSIF (rMetricIn < rMetricInMin) THEN
	rNumericOut := rNumericOutMin;
	bSignalStatus := 1;
ELSE
	bSignalStatus := 0;
END_IF

END_FUNCTION_BLOCK

// PFC200_CS_2ETH_RS_CAN_DPS/PFC8206/Scaling/fbScale_AI_457
FUNCTION_BLOCK fbScale_AI_457

VAR_INPUT

	rNumericIn: REAL;
	rMetricOutMin: REAL := -10;
	rMetricOutMax: REAL := 10;

END_VAR


VAR_OUTPUT

	rMetricOut: REAL;
	bSignalStatus : BYTE;

END_VAR


VAR

	LIN_TRAFO_ScaleAnalog: LIN_TRAFO;
	rNumericInMin: REAL := -32768;
	rNumericInMax: REAL := 32760;

END_VAR

LIN_TRAFO_ScaleAnalog(
	IN			:= rNumericIn,
	IN_MIN		:= rNumericInMin,
	IN_MAX		:= rNumericInMax,
	OUT_MIN		:= rMetricOutMin,
	OUT_MAX		:= rMetricOutMax,
	OUT			=> rMetricOut );


IF ( (REAL_TO_WORD(rNumericIn) AND 16#0003) > 0 ) THEN
	IF (REAL_TO_WORD(rNumericIn) > rNumericInMax) THEN
		rMetricOut := rMetricOutMax;
		bSignalStatus := 2;
	ELSE
		rMetricOut := rMetricOutMin;
		bSignalStatus := 1;
	END_IF
ELSE
	bSignalStatus := 0;
END_IF

END_FUNCTION_BLOCK

// PFC200_CS_2ETH_RS_CAN_DPS/PFC8206/Visu1
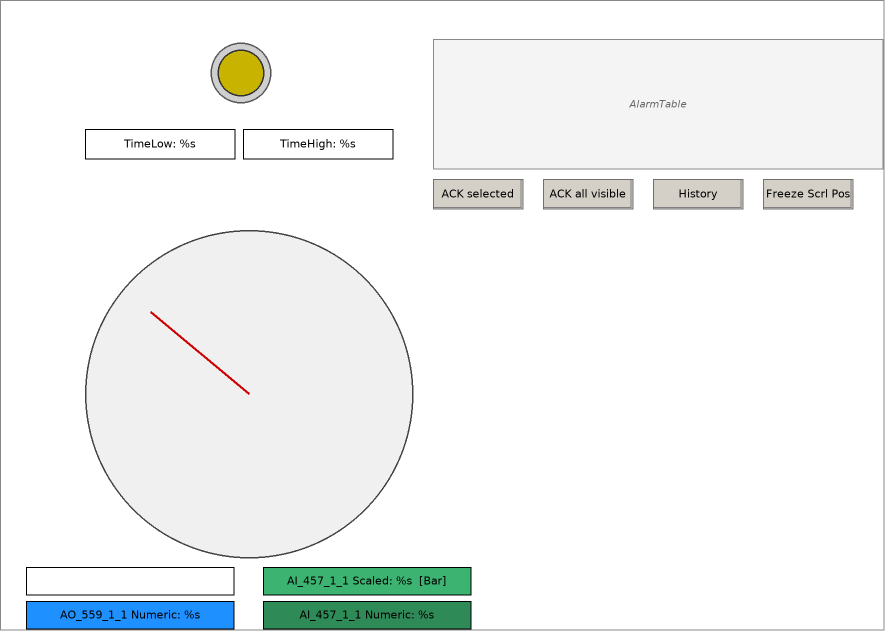
VISUALIZATION Visu1  // 885x631
VAR_IN_OUT
END_VAR
VAR
	bAckSel : BOOL;
	bAckVisible : BOOL;
	bHistory : BOOL;
	bFreezeScrlPos : BOOL;
END_VAR
    Lamp1 (206,38 70x70), variable: DO1, style: Lamp-Lamp1-Yellow
    Rectangle (85,129 150x30), "TimeLow: %s", text variable: PLC_PRG.tTimeLow
        OnMouseDown: write the text variable via Default
    Rectangle (243,129 150x30), "TimeHigh: %s", text variable: PLC_PRG.tTimeHigh
        OnMouseDown: write the text variable via Default
    Rectangle (26,567 208x28), "AO_559_1_1 Scaled: %s [rpm]", text variable: ScaleTest.AO_SpeedSet_1_Signal
        OnMouseDown: write the text variable via Edit
    Rectangle (263,567 208x28), "AI_457_1_1 Scaled: %s [Bar]", text variable: ScaleTest.AI_SpeedActual_1_Signal
    AlarmTable (433,39 450x130)
        Column[0]: ColumnTitle=Timestamp
        Column[1]: ColumnTitle=Message
        p1521930926: __All
        p1663851261: __All
        p428520879: bAckSel
        p2607059081: bAckVisible
        p3266827225: bHistory
        p3894972949: bFreezeScrlPos
    Button (433,179 90x30), "ACK selected"
        toggle bAckSel
    Button (543,179 90x30), "ACK all visible"
        toggle bAckVisible
    Button (653,179 90x30), "History"
        toggle bHistory
    Button (763,179 90x30), "Freeze Scrl Pos"
        toggle bFreezeScrlPos
    Meter360 (85,229 328x330), value: AO_559_1_1, style: Meter-Meter360-Gray, scale format: %.1f, scale 0..50000
    Rectangle (26,601 208x28), "AO_559_1_1 Numeric: %s", text variable: AO_559_1_1
    Rectangle (263,601 208x28), "AI_457_1_1 Numeric: %s", text variable: AI_457_1_1
END_VISUALIZATION

(* text list AlarmGroup1 (id | default)
  0 | MinAlarm1
   |  *)
